KUKA KRL data list: RoboSyncPidControl.dat

&ACCESS RVO3
&REL 16
&PARAM DISKPATH = KRC:\R1\TP\CNCRobotics\CEAD
DEFDAT  RoboSyncPidControl PUBLIC
;************************************************
;     NextState Automation Ltd
;     www.nextstateautomation.co.uk
;************************************************
;     Contact: helpdesk@nextstate.co.uk
;     Date: 14/09/26
;     Version: 0.1.1
;************************************************

GLOBAL ENUM ENUM_PID_TYPE HEATED_BED, EXTRUDER0, EXTRUDER1, NOZZLE

GLOBAL CONST INT AUTOTUNE_FAST=1
GLOBAL CONST INT AUTOTUNE_FULL=2
GLOBAL CONST INT AUTOTUNE_STOP=0

GLOBAL REAL pidDefaultUpperLimit=1.25
GLOBAL REAL pidDefaultLowerLimit=0.75

GLOBAL REAL rTemperatureTolerance = 10

GLOBAL CONST INT AUTOTUNE_TIMER=19
GLOBAL INT nAutotuneStartTimeout = 5000

ENDDAT
